FUNCTION Convert_LREAL_TO_STRING : Hresult
VAR_INPUT
	in : LREAL;
	out : REFERENCE TO STRING;
END_VAR
VAR
	converted : STRING;
END_VAR

converted := LREAL_TO_STRING(in);

IF (STRING_TO_LREAL(converted) <> in) THEN
	Convert_LREAL_TO_STRING := INCOMPATIBLE;
	RETURN;
END_IF

out := converted;

END_FUNCTION

(* stored: Version 1.1.0.1, ProductVersion 3.1.4024.12
   POU Convert_LREAL_TO_STRING: Id {857ccd25-a394-4109-ac51-6054e3df8112}, SpecialFunc None *)
